# EPICS substitutions: ek9000App/Db/EL3681.substitutions
file EL3681.template
{       pattern
        {
                TERMINAL,

        }
        {
        }
}
